FUNCTION_BLOCK Machine IMPLEMENTS IMachine
VAR_INPUT
END_VAR
VAR_OUTPUT
END_VAR
VAR
	Xts : XtsTrack;
	stateMachine : PMLStateMachine;
	indexMovers : ARRAY[1..10] OF IndexMover;
	Movers : ARRAY[1..10] OF IMover;
	StationArray : ARRAY[1..3] OF Station;
	iStationArray : ARRAY[1..3] OF IStation;
	i: INT;
	bInit: BOOL;
END_VAR

IF NOT bInit THEN
	FOR i := 1 TO 10 DO
		Movers[i] := indexMovers[i];
	END_FOR
	FOR i := 1 TO 3 DO
		iStationArray[i] := StationArray[i];
	END_FOR
	StationArray[1].Position := 1500.0;
	StationArray[2].Position := 2000.0;
	StationArray[3].Position := 2250.0;
	stateMachine.PMLCommand(Command := Tc3_PackML_V2.E_PMLState.ePMLState_Aborting);
	stateMachine.StateComplete();
	bInit := TRUE;
END_IF
stateMachine();
Xts(MoverArray := Movers, StateMachine := stateMachine);
FOR i := 1 TO 10 DO
	indexMovers[i](XtsTrack := Xts, StateMachine := stateMachine, StationArray := iStationArray );	
END_FOR

{warning 'add property implementation'}
PROPERTY PMLState : PackMLState
GET
//PMLState := State;
END_GET
END_PROPERTY

END_FUNCTION_BLOCK

(* stored: Version 1.1.0.1, ProductVersion 3.1.4024.9
   POU Machine: Id {e8d4edde-6e68-4e80-9f5b-2e9346044142}, SpecialFunc None
   Property PMLState: Id {ba36824d-caae-4e6e-b5dc-fb0feef88a75}
   Get Get: Id {ffdc919f-10da-4d02-addd-3d5827ea1ee1} *)
